TYPE ST_MOVER_OFFSETS :
STRUCT
  // static position offsets in stations
  PositionOffset      : ARRAY[1..MAX_STATION] OF T_NEST_OFFSET; // added to PosStop[] in XtsStation
END_STRUCT
END_TYPE

(* stored: Version 1.1.0.1, ProductVersion 3.1.4026.20
   DUT ST_MOVER_OFFSETS: Id {54474cd7-ae93-442f-b15d-5f6a7a65c69f} *)
